// TIA Portal V18 export
TYPE "StaProcessData"
// stored: IsFailsafeCompliant false
   STRUCT
      Reserved0 : Bool;   // 预留
      Reserved1 : Bool;   // 预留
      PartResult : Byte;   // 0-未作，1-合格，2-不合格
      PalletNo : Int;   // 托盘号
      Mode : Int;   // 作业模式
      PartID : String[48];   // 产品序列号
      "P-SubPartID" : Array[1..10] of String[48];   // 子零件号
   END_STRUCT;
END_TYPE
